// TIA Portal V20 export
DATA_BLOCK "DB_ToteTracking"   // DB15
// stored: MemoryReserve 100, Namespace ProductionLine
   VAR
      Conveyor : Array[_.minProductionLine.._.maxProductionLine] of "Global.TrackingData";
      Barcode : Array[_.minProductionLine.._.maxProductionLine] of String;
      Transfer : Array[_.minProductionLine.._.maxProductionLine] of "Global.ItemDir";
   END_VAR
BEGIN
END_DATA_BLOCK
